Staubli VAL3: sendCommand.pgx

program sendCommand(num handle_, string cmd_, bool& result_[])
  local string msg
  local bool dummy
  local string str
begin
  // send native command to camera and read command execution result
  call writeSocket(handle_,cmd_)
  call readSocket(handle_,msg,result_)
  str=toNum(msg,errorCode[handle_],dummy)
  result_=errorCode[handle_]==1
  if bDebug
    call getErrorMessage(handle_,msg)
    putln("result: "+msg)
  endIf
end
